FUNCTION_BLOCK AROBOT_DEMUX (* Composite FB wrapping other FBs *)
  (* Standard: 61499-2 *)
  (* Version 0.0, 2008-07-10, 4DIAC-IDE, 4DIAC-Consortium *)
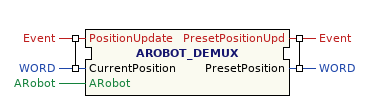
  EVENT_INPUT
    PositionUpdate WITH CurrentPosition; (* Request from Socket *)
  END_EVENT
  EVENT_OUTPUT
    PresetPositionUpd WITH PresetPosition; (* Indication from Plug *)
  END_EVENT
  VAR_INPUT
    CurrentPosition : WORD; (* Request Data from Socket *)
  END_VAR
  VAR_OUTPUT
    PresetPosition : WORD; (* Confirmation Data from Plug *)
  END_VAR
  SOCKETS
    ARobot : ARobot;
  END_SOCKETS
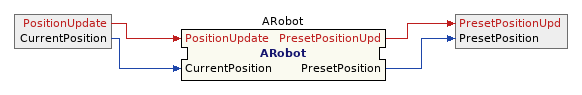
  EVENT_CONNECTIONS
    PositionUpdate TO ARobot.PositionUpdate;
    ARobot.PresetPositionUpd TO PresetPositionUpd;
  END_CONNECTIONS
  DATA_CONNECTIONS
    CurrentPosition TO ARobot.CurrentPosition;
    ARobot.PresetPosition TO PresetPosition;
  END_CONNECTIONS
END_FUNCTION_BLOCK
